TEXTLIST ActionMode
  1 = '直線動作(MoveToPosition)'
  2 = '回転動作(MoveC)'
  3 = '上下動作(MoveZ)'
  4 = '前後動作(MoveA)'
  5 = '左右動作(MoveB)'
  6 = '前後左右(MoveA/B混合)'
   = ''
END_TEXTLIST

(* stored: Version 1.1.0.1, ProductVersion 3.1.4024.12
   TextList ActionMode: Id {da26fca6-735d-4f7a-ba7b-44acea908699} *)
